FUNCTION_BLOCK "LVT_ModbusDeviceRtu_Master"
{ S7_Optimized_Access := 'TRUE' }
AUTHOR : 'Anatoly Veshtemov'
FAMILY : LVT
   VAR_INPUT
      start : Bool;   // Start block
   END_VAR

   VAR_OUTPUT
      busy { ExternalWritable := 'False'} : Bool;   // In progress
      done { ExternalWritable := 'False'} : Bool;   // Done
   END_VAR

   VAR_IN_OUT
      readBuffer : Variant;   // Pointer of read buffer (non optimized data block). For example, DB -> readBuffer: Array[0..125] of Word
      writeBuffer : Variant;   // Pointer of write buffer (non optimized data block). For example, DB -> writeBuffer: Array[0..125] of Word
      data : "LVT_typeModbusDeviceRtu_Data";
      mbMaster {InstructionName := 'Modbus_Master'; LibVersion := '3.2'} : Modbus_Master;   // Instance of Modbus_Master function block
   END_VAR

   VAR
      statBuffer : Array[0..127] of Word;
      startTrig {InstructionName := 'R_TRIG'; LibVersion := '1.0'; ExternalAccessible := 'False'; ExternalVisible := 'False'; ExternalWritable := 'False'; S7_SetPoint := 'False'} : R_TRIG;   // Detect start
      statWatchdogTimer {InstructionName := 'TON_TIME'; LibVersion := '1.0'; ExternalAccessible := 'False'; ExternalVisible := 'False'; ExternalWritable := 'False'; S7_SetPoint := 'False'} : TON_TIME;   // Timer for resetting a request when unknown reason is happened
      statState { ExternalAccessible := 'False'; ExternalVisible := 'False'; ExternalWritable := 'False'} : USInt;   // Current state
      i { ExternalAccessible := 'False'; ExternalVisible := 'False'; ExternalWritable := 'False'} : Int;
      j { ExternalAccessible := 'False'; ExternalVisible := 'False'; ExternalWritable := 'False'} : Int;
   END_VAR

   VAR_TEMP
      tempStart : Bool;   // Start flag
      tempRetval : Int;
      tempQntRequests : Int;   // Quantity of requests
      tempZeroIndex : DInt;
   END_VAR

   VAR CONSTANT
      STATE_STANDBY : USInt := 0;   // State. Standby
      STATE_SETTINGS : USInt := 1;   // State. Get settings
      STATE_READ : USInt := 2;   // State. Reading
      STATE_WRITE : USInt := 3;   // State. Writing
      STATE_HANDLE : USInt := 4;   // State. Handle results
      WATCHDOG_TIME : Time := T#10S;   // Watchdog time
      ERROR_ILLEGAL_REQUEST : Word := 16#9000;   // Error. Illegal request (check request settings)
      ERROR_WATCHDOG_TIMER : Word := 16#9001;   // Error. Watchdog timer
   END_VAR


BEGIN
	REGION Block info header
	    //===============================================================================
	    // (company) / (c)Copyright year
	    //-------------------------------------------------------------------------------
	    // Title:            LVT_ModbusDevcieRtu_Master
	    // Comment/Function: Modbus RTU Master device-oriented
	    //                   Requests are grouped for each network device separately, and devices are sequentially polled.
	    //                   Each network device has a local data buffer.
	    // Library/Family:   LVT
	    // Author:           Anatoly Veshtemov
	    // Tested with:      CPU 1214C
	    // Engineering:      TIA Portal V17
	    // Restrictions:     no
	    // Requirements:     PLC (S7-1200 / S7-1500)
	    //-------------------------------------------------------------------------------
	    // Change log table:
	    // Version  | Date       | Expert in charge       | Changes applied
	    //----------|------------|------------------------|------------------------------
	    // 00.00.04 01.01.2023  First released version
	    // 00.01.00 17.06.2026  Upgrate to TIA V17
	    //                      Added block info header
	    //                      Refactor names in Static
	    //=============================================================================

	END_REGION Block info header

	REGION DESCRIPTION
	    (/**/)
	END_REGION DESCRIPTION

	#tempQntRequests := UDINT_TO_INT("LVT_ModbusDeviceRtu_GetArrayLength"(arr := #data.requests));
	#busy := (#statState > #STATE_STANDBY); // Set busy flag

	#startTrig(CLK := #start,
	                Q => #tempStart);

	// When start go to Settings
	IF #tempStart THEN

	    #done := false;
	    #statState := #STATE_SETTINGS;

	END_IF;

	CASE #statState OF

	        // Standby
	    #STATE_STANDBY:

	        #done := false;
	        #i := 0;

	        // Get request settings
	    #STATE_SETTINGS:

	        // With the first call we reset the counter, get the first request,
	        // else we increase counter by 1 and get a next request
	        IF #tempStart THEN
	            #i := 0;

	        ELSE
	            #i := #i + 1;

	            // When all requests is completed go to standby, set "done" flag
	            IF #i >= #tempQntRequests THEN
	                #done := true;
	                #statState := #STATE_STANDBY;
	                RETURN;
	            END_IF;
	        END_IF;

	        // Check request settings: we have to skip disabled or invalid requests,
	        // if a request is invalid - set ERROR_ILLEGAL_REQUEST status
	        FOR #j := #i TO #tempQntRequests - 1 DO

	            IF NOT #data.requests[#j].cfg.enable THEN

	                #data.requests[#j].status.req := false;
	                #data.requests[#j].status.done := false;
	                #data.requests[#j].status.error := false;
	                #data.requests[#j].status.status := 0;
	                #data.requests[#j].status.errorCounter := 0;

	            ELSIF NOT "LVT_ModbusDeviceRtu_ValidateRequest"(data := #data, index := #j) THEN

	                // Set error status
	                #data.requests[#j].status.req := false;
	                #data.requests[#j].status.done := false;
	                #data.requests[#j].status.error := true;
	                #data.requests[#j].status.status := #ERROR_ILLEGAL_REQUEST;
	                #data.requests[#j].status.errorCounter := LIMIT(IN := #data.requests[#j].status.errorCounter + 1,
	                                                                MN := 0,
	                                                                MX := 65534);
	            ELSE
	                #i := #j;
	                EXIT;
	            END_IF;

	            // When all requests is completed go to standby, set "done" flag
	            IF #j = #tempQntRequests - 1 THEN
	                #done := true;
	                #statState := #STATE_STANDBY;
	                RETURN;
	            END_IF;

	        END_FOR;

	        // For writing before request we have to copy data to external write buffer
	        IF #data.requests[#i].cfg.mode > 0 THEN

	            // Extract data from Modbus Device to write buffer
	            MOVE_BLK(IN := #data.#buffer[#data.requests[#i].cfg.mapAddr],
	                     COUNT := #data.requests[#i].cfg.len,
	                     OUT => #statBuffer[0]);

	            #tempZeroIndex := 0;
	            #tempRetval := Serialize(SRC_VARIABLE := #statBuffer,
	                                     DEST_ARRAY => #writeBuffer,
	                                     POS := #tempZeroIndex);

	            #statState := #STATE_WRITE;
	        ELSE
	            #statState := #STATE_READ;
	        END_IF;

	        RETURN;

	        // Read
	    #STATE_READ, #STATE_WRITE:

	        #data.requests[#i].status.req := true;

	        // Handle results
	    #STATE_HANDLE:

	        #data.requests[#i].status.req := false;

	        IF #data.requests[#i].status.done THEN
	            #data.requests[#i].status.errorCounter := 0;

	            // Copy from modbus buffer to device buffer
	            IF #data.requests[#i].cfg.mode = 0 THEN

	                #tempZeroIndex := 0;
	                #tempRetval := Deserialize(SRC_ARRAY := #readBuffer,
	                                           DEST_VARIABLE => #statBuffer,
	                                           POS := #tempZeroIndex);
	                MOVE_BLK(IN := #statBuffer[0],
	                         COUNT := #data.requests[#i].cfg.len,
	                         OUT => #data.buffer[#data.requests[#i].cfg.mapAddr]);
	            END_IF;

	        ELSIF #data.requests[#i].status.error THEN
	            #data.requests[#i].status.errorCounter := LIMIT(IN := #data.requests[#i].status.errorCounter + 1,
	                                                            MN := 0,
	                                                            MX := 65534);
	        END_IF;

	        #statState := #STATE_SETTINGS;

	    ELSE
	        #statState := #STATE_STANDBY;
	END_CASE;

	// There are different buffers for reading and writing
	IF (#statState = #STATE_READ) THEN
	    // Request
	    #mbMaster(REQ := #data.requests[#i].status.req,
	              MB_ADDR := #data.address,
	              MODE := #data.requests[#i].cfg.mode,
	              DATA_ADDR := #data.requests[#i].cfg.dataAddr,
	              DATA_LEN := #data.requests[#i].cfg.len,
	              DONE => #data.requests[#i].status.done,
	              BUSY => #data.requests[#i].status.busy,
	              ERROR => #data.requests[#i].status.error,
	              STATUS => #data.requests[#i].status.status,
	              DATA_PTR := #readBuffer);

	ELSIF (#statState = #STATE_WRITE) THEN
	    // Request
	    #mbMaster(REQ := #data.requests[#i].status.req,
	              MB_ADDR := #data.address,
	              MODE := #data.requests[#i].cfg.mode,
	              DATA_ADDR := #data.requests[#i].cfg.dataAddr,
	              DATA_LEN := #data.requests[#i].cfg.len,
	              DONE => #data.requests[#i].status.done,
	              BUSY => #data.requests[#i].status.busy,
	              ERROR => #data.requests[#i].status.error,
	              STATUS => #data.requests[#i].status.status,
	              DATA_PTR := #writeBuffer);
	END_IF;


	// Waiting response status
	IF ((#statState = #STATE_READ
	    OR #statState = #STATE_WRITE)
	    AND (#data.requests[#i].status.done
	    OR #data.requests[#i].status.error))
	THEN
	    #statState := #STATE_HANDLE;
	END_IF;

	// Watchdog timer is needed when state stuck in Read or Write state for unknown reason,
	// in that case we set request as invalid
	#statWatchdogTimer(IN := (#statState = #STATE_READ
	                    OR #statState = #STATE_WRITE),
	                    PT := #WATCHDOG_TIME);

	IF #statWatchdogTimer.Q THEN

	    #data.requests[#i].status.done := false;
	    #data.requests[#i].status.error := true;
	    #data.requests[#i].status.status := #ERROR_WATCHDOG_TIMER;
	    #data.requests[#i].status.errorCounter := LIMIT(IN := #data.requests[#i].status.errorCounter + 1,
	                                                    MN := 0,
	                                                    MX := 65534);

	    #statState := #STATE_HANDLE;

	END_IF;
END_FUNCTION_BLOCK

